{attribute 'qualified_only'}
{attribute 'strict'}
{attribute 'to_string'}
TYPE TIMESTAMP_DISPLAY_MODE :
(
	HIDDEN := 0,
	LOCAL, 
	UTC
);
END_TYPE

(* stored: Version 1.1.0.1
   DUT TIMESTAMP_DISPLAY_MODE: Id {c51f99b6-5d13-4a9d-9983-9a3a07f2fd1e} *)
